INTERFACE I_HE_SATT_FilterWedge EXTENDS I_HE_SATT_Filter


METHOD ThicknessAt : LREAL
VAR_INPUT
    fPosition : LREAL; // Position in units of property Length and with value from 0 to value of property Length
END_VAR
END_METHOD

END_INTERFACE

(* stored: Version 1.1.0.1
   Itf I_HE_SATT_FilterWedge: Id {07fda710-a856-45c4-9342-2b90967d8a83}
   Method ThicknessAt: Id {81688184-8feb-4b22-ab03-0cd1e3659053} *)
